FUNCTION_BLOCK EMB_RES
  {SET_ATTRIBUTE(OpcUa, DEVICE.SENSOR)}
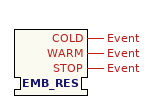
  EVENT_OUTPUT
    COLD;
    WARM;
    STOP;
  END_EVENT
END_FUNCTION_BLOCK
